FUNCTION TryConvert_INT_TO_TIME : BOOL
VAR_INPUT
	in : INT;
	out : REFERENCE TO TIME;
END_VAR

IF in < DatatypeLimits.MIN_VALUE_OF_INT_WHICH_CAN_BE_HELD_IN_A_TIME THEN
	RETURN;
END_IF

out := INT_TO_TIME(in);
TryConvert_INT_TO_TIME := TRUE;

END_FUNCTION

(* stored: Version 1.1.0.1, ProductVersion 3.1.4024.12
   POU TryConvert_INT_TO_TIME: Id {fece783a-ca47-4cd4-933c-ec738c4a8783}, SpecialFunc None *)
